TYPE ST_SelectorM3 EXTENDS ST_Selector :
STRUCT
	//Flowmeters
	////////////////////////
		stMFM	:	ST_BhElFlow;
		astSelFM	: ARRAY[1..2] OF	ST_SensirionFM; //Address 1 is low flow, address 2 is high flow, low flow is mapped to M2 flow
		fbSensirionDriver	:	ARRAY [1..2] OF	FB_SensirionDriver;
		
		rLowFlow	:	REAL;
		rHighFlow	:	REAL;
		rGasFlow	:	REAL; //El-flow
END_STRUCT
END_TYPE

(* stored: Version 1.1.0.1, ProductVersion 3.1.4018.5
   DUT ST_SelectorM3: Id {fa3c6e97-4043-47eb-be01-712b94ca71b0} *)
